// TwinCAT 3 PLC project SPS
// ProgramVersion: 3.1.4024.0
// libraries:
//   Tc2_MC2, * (Beckhoff Automation GmbH)
//   Tc2_Standard, * (Beckhoff Automation GmbH)
//   Tc2_System, * (Beckhoff Automation GmbH)
//   Tc3_IotBase, * (Beckhoff Automation GmbH)
//   Tc3_Module, * (Beckhoff Automation GmbH)
// project tree:
//   DUTs/ eBetriebszustand.TcDUT
//   GVLs/ GVL_PosKinematic.TcGVL, IFC_HW.TcGVL (not stored)
//   / PlcTask.TcTTO
//   POUs/Abfüllmodul/Ampelleuchte/ FB_Ampelstatus.TcPOU (not stored), FB_Blinklicht.TcPOU
//   POUs/Abfüllmodul/ FB_Abfullmodul.TcPOU, FB_Dispenser.TcPOU
//   POUs/Abfüllmodul/Tranport/ FB_Forderband.TcPOU, FB_Transport.TcPOU, FB_TransportA.TcPOU (not stored), FB_TransportE.TcPOU, FB_TransportLogik.TcPOU
//   POUs/Abfüllmodul/Vereinzelung/ FB_EZylinder.TcPOU (not stored), FB_Vereinzelung.TcPOU (not stored)
//   POUs/ FB_Maschinentuer.TcPOU, FB_Testmaschinentuer.TcPOU, MAIN.TcPOU, FUN_linear_Scale.TcPOU
//   POUs/IOT/ FB_MqttClient.TcPOU
//   POUs/Robotermodul/ FB_Roboterablauf.TcPOU, FB_Robotersteuerung.TcPOU, FB_Roboterachsensteuerung.TcPOU
// real-time tasks:
//   TASK PlcTask: cycle T#10ms, priority 20, ADS port 350
// motion (NC):
//   TASK NC-Task 1 SAF: cycle T#2ms, priority 4, ADS port 501
//   TASK NC-Task 1 SVB: cycle T#10ms, priority 8, ADS port 511
//   AXIS Achse_Band (id 1)
//     OtherSettings: AllowMotionCmdToSlave=true
//     encoder EncType=1
//     drive DrvType=5
//       Analog: TorqueSetpointScale=10, ScaleFactorActTorque=0.1
//       TimeComp: TaskDelayCycles=1
//     controller CtrType=1
//       CtrPara: PriorControlFactor=1
//         Observer: BandWidth=20
//   AXIS Achse_Extruder1 (id 2)
//     OtherSettings: AllowMotionCmdToSlave=true
//     encoder EncType=1
//     drive DrvType=5
//       Analog: TorqueSetpointScale=10, ScaleFactorActTorque=0.1
//       TimeComp: TaskDelayCycles=1
//     controller CtrType=1
//       CtrPara: PriorControlFactor=1
//         Observer: BandWidth=20
//   AXIS Achse_Extruder2 (id 3)
//     OtherSettings: AllowMotionCmdToSlave=true
//     encoder EncType=1
//     drive DrvType=5
//       Analog: TorqueSetpointScale=10, ScaleFactorActTorque=0.1
//       TimeComp: TaskDelayCycles=1
//     controller CtrType=1
//       CtrPara: PriorControlFactor=1
//         Observer: BandWidth=20
//   AXIS Achse_Extruder3 (id 4)
//     OtherSettings: AllowMotionCmdToSlave=true
//     encoder EncType=1
//     drive DrvType=5
//       Analog: TorqueSetpointScale=10, ScaleFactorActTorque=0.1
//       TimeComp: TaskDelayCycles=1
//     controller CtrType=1
//       CtrPara: PriorControlFactor=1
//         Observer: BandWidth=20
//   AXIS Roboter_x (id 5)
//     OtherSettings: AllowMotionCmdToSlave=true
//     encoder EncType=1
//       EncPara: ScaleFactorNumerator=1
//         Inc: RefSearchInverse=true, RefSyncInverse=false
//     drive DrvType=5
//       Analog: TorqueSetpointScale=10, ScaleFactorActTorque=0.1
//       TimeComp: TaskDelayCycles=1
//     controller CtrType=1
//       CtrPara: PriorControlFactor=1
//         Observer: BandWidth=20
//   AXIS Roboter_y (id 6)
//     OtherSettings: AllowMotionCmdToSlave=true
//     encoder EncType=1
//       EncPara: ScaleFactorNumerator=1
//         Inc: RefSearchInverse=true, RefSyncInverse=false
//     drive DrvType=5
//       Analog: TorqueSetpointScale=10, ScaleFactorActTorque=0.1
//       TimeComp: TaskDelayCycles=1
//     controller CtrType=1
//       CtrPara: PriorControlFactor=1
//         Observer: BandWidth=20
//   AXIS Roboter_z (id 7)
//     OtherSettings: AllowMotionCmdToSlave=true
//     encoder EncType=1
//       EncPara: ScaleFactorNumerator=1
//         Inc: RefSearchInverse=true, RefSyncInverse=false
//     drive DrvType=5
//       Analog: TorqueSetpointScale=10, ScaleFactorActTorque=0.1
//       TimeComp: TaskDelayCycles=1
//     controller CtrType=1
//       CtrPara: PriorControlFactor=1
//         Observer: BandWidth=20
//   AXIS Roboter_g (id 8)
//     OtherSettings: AllowMotionCmdToSlave=true
//     encoder EncType=1
//       EncPara: ScaleFactorNumerator=1
//     drive DrvType=5
//       Analog: TorqueSetpointScale=10, ScaleFactorActTorque=0.1
//       TimeComp: TaskDelayCycles=1
//     controller CtrType=1
//       CtrPara: PriorControlFactor=1
//         Observer: BandWidth=20
// variable links:
//   SPS/SPS Instance <-> NC-Task 1 SAF/Axes/Achse_Band
//     PlcTask Inputs/IFC_HW.ax_BandMotor.NcToPlc <-> Outputs/ToPlc
//     PlcTask Outputs/IFC_HW.ax_BandMotor.PlcToNc <-> Inputs/FromPlc
//   SPS/SPS Instance <-> NC-Task 1 SAF/Axes/Achse_Extruder1
//     PlcTask Inputs/IFC_HW.ax_Extruder1.NcToPlc <-> Outputs/ToPlc
//     PlcTask Outputs/IFC_HW.ax_Extruder1.PlcToNc <-> Inputs/FromPlc
//   SPS/SPS Instance <-> NC-Task 1 SAF/Axes/Achse_Extruder2
//     PlcTask Inputs/IFC_HW.ax_Extruder2.NcToPlc <-> Outputs/ToPlc
//     PlcTask Outputs/IFC_HW.ax_Extruder2.PlcToNc <-> Inputs/FromPlc
//   SPS/SPS Instance <-> NC-Task 1 SAF/Axes/Achse_Extruder3
//     PlcTask Inputs/IFC_HW.ax_Extruder3.NcToPlc <-> Outputs/ToPlc
//     PlcTask Outputs/IFC_HW.ax_Extruder3.PlcToNc <-> Inputs/FromPlc
//   SPS/SPS Instance <-> NC-Task 1 SAF/Axes/Roboter_g
//     PlcTask Inputs/IFC_HW.ax_ManG.NcToPlc <-> Outputs/ToPlc
//     PlcTask Outputs/IFC_HW.ax_ManG.PlcToNc <-> Inputs/FromPlc
//   SPS/SPS Instance <-> NC-Task 1 SAF/Axes/Roboter_x
//     PlcTask Inputs/IFC_HW.ax_ManX.NcToPlc <-> Outputs/ToPlc
//     PlcTask Outputs/IFC_HW.ax_ManX.PlcToNc <-> Inputs/FromPlc
//   SPS/SPS Instance <-> NC-Task 1 SAF/Axes/Roboter_y
//     PlcTask Inputs/IFC_HW.ax_ManY.NcToPlc <-> Outputs/ToPlc
//     PlcTask Outputs/IFC_HW.ax_ManY.PlcToNc <-> Inputs/FromPlc
//   SPS/SPS Instance <-> NC-Task 1 SAF/Axes/Roboter_z
//     PlcTask Inputs/IFC_HW.ax_ManZ.NcToPlc <-> Outputs/ToPlc
//     PlcTask Outputs/IFC_HW.ax_ManZ.PlcToNc <-> Inputs/FromPlc

CONFIGURATION SPS
    RESOURCE PLC ON TwinCAT3
        TASK PlcTask(INTERVAL := T#10ms, PRIORITY := 20);
        PROGRAM MAIN WITH PlcTask : MAIN;
    END_RESOURCE
END_CONFIGURATION

// ---- DUTs/eBetriebszustand.TcDUT
{attribute 'qualified_only'}
{attribute 'strict'}
TYPE eBetriebszustand :
(
	WARNING,	// Nicht fehlerbehafteter/ungeplanter Stop
	ERROR,		// Fehlerbehafteter Stop
	STOP,		// Geplanter Stop
	OFF,		// Nicht Betriebsbereit
	INIT,		// Herstellung betriebsbereit
	PROD,		// Betrieb
	READY,		// Betriebsbereit
	DONE,		// Betrieb abgeschlosen
	SETUP		// Wartung
);
END_TYPE

// ---- GVLs/GVL_PosKinematic.TcGVL
{attribute 'qualified_only'}
VAR_GLOBAL
	// Home position
	pXhome : REAL := 29;
	pYhome : REAL := 145.5;
	pZhome : REAL := 45;
	
	// Conveyor position
	pXconv : REAL := 29;
	pYconv : REAL := 145.5;
	pZconv : REAL := 130;
	
	// Scale position
	pXscale : REAL := 36;
	pYscale : REAL := 7.5;
	pZscale : REAL := 131.5;
	
	// Heating position
	pXheat : REAL := 218.5;
	pYheat : REAL := 7;
	pZheat : REAL := 159;
	
	// Storage position
	pX1stor : REAL := 107;
	pX2stor : REAL := 158.7;
	pX3stor : REAL := 209.3;
	pX4stor : REAL := 260.3;
	pYstor : REAL := 139;
	pZstor : REAL := 120;
	
	// Z offset height
	pZoff : REAL := 45;
END_VAR

// ---- POUs/MAIN.TcPOU
PROGRAM MAIN
VAR
	fbAbfullmodul : FB_Abfullmodul;
	fbStatusAmpel : FB_Ampelstatus;
	fbRoboter : FB_Roboterablauf;
	fbMqttClient : FB_MqttClient;
END_VAR

fbAbfullmodul(
	bEnable:= IFC_HW.bEnable, 
	bExecute:= IFC_HW.bExecute, 
	eState=> fbStatusAmpel.eState, 
	ax1:= IFC_HW.ax_Extruder1, 
	ax2:= IFC_HW.ax_Extruder2, 
	ax3:= IFC_HW.ax_Extruder3);
	
fbStatusAmpel(
	eState:= , 
	bLightRed=> IFC_HW.bAmpelRot, 
	bLightYellow=> IFC_HW.bAmpelGelb, 
	bLightGreen=> IFC_HW.bAmpelGrun);
	
fbRoboter(bEnable:= IFC_HW.bEnable, bExecute:= IFC_HW.bBandSens4, eState=> );

fbMqttClient();

END_PROGRAM

// ---- POUs/Abfüllmodul/FB_Abfullmodul.TcPOU
FUNCTION_BLOCK FB_Abfullmodul
VAR_INPUT
    bEnable: BOOL;
    bExecute : BOOL;
END_VAR
VAR_OUTPUT
    eState : eBetriebszustand;
END_VAR
VAR
    nState : INT := 0;
    nStation :INT := 0;
    
    fbVereinzelung : FB_Vereinzelung;
    fbTransport : FB_Transport;
    fbDispenser1 : FB_Dispenser;
    fbDispenser2 : FB_Dispenser;
    fbDispenser3 : FB_Dispenser;
	fbEZylinder1: FB_EZylinder;
	fbEZylinder2: FB_EZylinder;
END_VAR
VAR_IN_OUT
    ax1 : AXIS_REF;
	ax2 : AXIS_REF;
	ax3 : AXIS_REF;
END_VAR

fbVereinzelung(
	bEnable:= bEnable, 
	bExecute:= , 
	bSensor1:= IFC_HW.bEinzelSens1, 
	bSensor2:= IFC_HW.bEinzelSens2, 
	bSensor3:= IFC_HW.bEinzelSens3, 
	bSensor4:= IFC_HW.bBandSens1, 
	eState=> , 
	bGate1=> fbEZylinder1.bGate, 
	bGate2=> fbEZylinder2.bGate);
	
fbEZylinder1(bGate:= , bError:= , bR1=> IFC_HW.bR1AKT1, bR2=> IFC_HW.bR2AKT1);
fbEZylinder2(bGate:= , bError:= , bR1=> IFC_HW.bR1AKT2, bR2=> IFC_HW.bR2AKT2);

fbTransport(
	bEnable:= bEnable, 
	bExecute:= , 
	nStation:= nStation, 
	bSens1:= IFC_HW.bBandSens1, 
	bSens2:= IFC_HW.bBandSens2, 
	bSens3:= IFC_HW.bBandSens3, 
	bSens4:= IFC_HW.bBandSens4, 
	eState=> , 
	bStopper1=> IFC_HW.bBandHub1, 
	bStopper2=> IFC_HW.bBandHub2, 
	bStopper3=> IFC_HW.bBandHub3, 
	ax:= IFC_HW.ax_BandMotor);
	
fbDispenser1(
	bEnable:= bEnable, 
	bExecute:= , 
	rDistance:= 100, 
	eState=> , 
	ax:= ax1);

fbDispenser2(
	bEnable:= bEnable, 
	bExecute:= , 
	rDistance:= 100, 
	eState=> , 
	ax:= ax2);

fbDispenser3(
	bEnable:= bEnable, 
	bExecute:= , 
	rDistance:= 100, 
	eState=> , 
	ax:= ax3);

CASE nState OF
	
	0: // OFF
	eState := eBetriebszustand.OFF;
	
	fbVereinzelung.bEnable := FALSE;
	fbTransport.bEnable := FALSE;
	fbDispenser1.bEnable := FALSE;
	fbDispenser2.bEnable := FALSE;
	fbDispenser3.bEnable := FALSE;
	
	fbVereinzelung.bExecute := FALSE;
	fbTransport.bExecute := FALSE;
	fbDispenser1.bExecute := FALSE;
	fbDispenser2.bExecute := FALSE;
	fbDispenser3.bExecute := FALSE;
	
	IF bEnable THEN
		nState:= 10; // INIT
	END_IF
	
	10: // INIT
	eState := eBetriebszustand.INIT;
	
	fbVereinzelung.bEnable := TRUE;
	fbTransport.bEnable := TRUE;
	fbDispenser1.bEnable := TRUE;
	fbDispenser2.bEnable := TRUE;
	fbDispenser3.bEnable := TRUE;
	
	fbVereinzelung.bExecute := FALSE;
	fbTransport.bExecute := FALSE;
	fbDispenser1.bExecute := FALSE;
	fbDispenser2.bExecute := FALSE;
	fbDispenser3.bExecute := FALSE;
	
	IF (fbVereinzelung.eState = eBetriebszustand.READY) AND (fbTransport.eState = eBetriebszustand.READY) AND (fbDispenser1.eState = eBetriebszustand.READY) 
		AND (fbDispenser2.eState = eBetriebszustand.READY) AND (fbDispenser3.eState = eBetriebszustand.READY) THEN
		
		nState := 20; // READY
	END_IF
	
	20: // READY
	eState := eBetriebszustand.READY;
	
	fbVereinzelung.bEnable := TRUE;
	fbTransport.bEnable := TRUE;
	fbDispenser1.bEnable := TRUE;
	fbDispenser2.bEnable := TRUE;
	fbDispenser3.bEnable := TRUE;
	
	IF bExecute THEN
		nState := 30; //Start
	END_IF
	
	30: // PROD - Start
	eState := eBetriebszustand.PROD;
	nStation := 1;
	
	fbVereinzelung.bEnable := TRUE;
	fbTransport.bEnable := TRUE;
	fbDispenser1.bEnable := TRUE;
	fbDispenser2.bEnable := TRUE;
	fbDispenser3.bEnable := TRUE;
	
	fbVereinzelung.bExecute := TRUE;
	fbTransport.bExecute := TRUE;
	fbDispenser1.bExecute := FALSE;
	fbDispenser2.bExecute := FALSE;
	fbDispenser3.bExecute := FALSE;
	
	IF (fbVereinzelung.eState = eBetriebszustand.DONE) AND (fbTransport.eState = eBetriebszustand.DONE)THEN
		nState := 31; // Extruder 1
	END_IF
	
	31: // PROD - Extruder 1
	eState := eBetriebszustand.PROD;
	nStation := 1;

	fbVereinzelung.bExecute := FALSE;
	fbTransport.bExecute := FALSE;
	fbDispenser1.bExecute := TRUE;
	fbDispenser2.bExecute := FALSE;
	fbDispenser3.bExecute := FALSE;
	
	IF fbDispenser1.eState = eBetriebszustand.DONE THEN
		nState := 32; // Bewegung zu Station 2
	END_IF
	
	32: // PROD - Bewegung zu Station 2
	eState := eBetriebszustand.PROD;
	nStation := 2;
	
	fbVereinzelung.bExecute := FALSE;
	fbTransport.bExecute := TRUE;
	fbDispenser1.bExecute := FALSE;
	fbDispenser2.bExecute := FALSE;
	fbDispenser3.bExecute := FALSE;
	
	IF fbTransport.eState = eBetriebszustand.DONE THEN
		nState := 33; //  Extruder 2
	END_IF
	
	33: // PROD - Extruder 2
	eState := eBetriebszustand.PROD;
	nStation := 2;
	
	fbVereinzelung.bExecute := FALSE;
	fbTransport.bExecute := FALSE;
	fbDispenser1.bExecute := FALSE;
	fbDispenser2.bExecute := TRUE;
	fbDispenser3.bExecute := FALSE;
	
	IF fbDispenser2.eState = eBetriebszustand.DONE THEN
		nState := 34; // Bewegung zu Station 3
	END_IF
	
	34: // PROD - Bewegung zu Station 3
	eState := eBetriebszustand.PROD;
	nStation := 3;
	
	fbVereinzelung.bExecute := FALSE;
	fbTransport.bExecute := TRUE;
	fbDispenser1.bExecute := FALSE;
	fbDispenser2.bExecute := FALSE;
	fbDispenser3.bExecute := FALSE;
	
	IF fbTransport.eState = eBetriebszustand.DONE THEN
		nState := 35; // Extruder 3
	END_IF
	
	35: // PROD - Extruder 3
	eState := eBetriebszustand.PROD;
	nStation := 3;
	
	fbVereinzelung.bExecute := FALSE;
	fbTransport.bExecute := FALSE;
	fbDispenser1.bExecute := FALSE;
	fbDispenser2.bExecute := FALSE;
	fbDispenser3.bExecute := TRUE;
	
	IF fbDispenser3.eState = eBetriebszustand.DONE THEN
		nState := 36; // Bewegung zu Abholstation
	END_IF
	
	36: // PROD - Bewegung zu Abholstation
	eState := eBetriebszustand.PROD;
	nStation := 4;
	
	fbVereinzelung.bExecute := FALSE;
	fbTransport.bExecute := TRUE;
	fbDispenser1.bExecute := FALSE;
	fbDispenser2.bExecute := FALSE;
	fbDispenser3.bExecute := FALSE; 
	
	IF fbTransport.eState = eBetriebszustand.DONE THEN
		nState := 40; // DONE
	END_IF
	
	40: // DONE
	eState :=  eBetriebszustand.DONE;
	nStation := 4;
	
	fbTransport.bExecute := False;
	
	IF NOT bExecute THEN
		nState := 20; // READY
	ELSIF nStation = 4 THEN
		nState := 30; // START
	END_IF
	
END_CASE

END_FUNCTION_BLOCK

// ---- POUs/Abfüllmodul/Tranport/FB_Transport.TcPOU
FUNCTION_BLOCK FB_Transport
VAR_INPUT
	bEnable : BOOL;
	bExecute : BOOL;
	nStation : INT;
	
	bSens1 : BOOL;
	bSens2 : BOOL;
	bSens3 : BOOL;
	bSens4 : BOOL;
END_VAR
VAR_OUTPUT
	eState : eBetriebszustand;
	
	bStopper1 : BOOL;
	bStopper2 : BOOL;
	bStopper3 : BOOL;
END_VAR
VAR
	fbTransportE : FB_TransportE;
	fbTransportLogik : FB_TransportLogik;
	fbTransportBand : FB_Forderband;
	fbTransportA : FB_TransportA;
END_VAR
VAR_IN_OUT
    ax : AXIS_REF;
END_VAR

fbTransportE(
	bSens1:= bSens1, 
	bSens2:= bSens2, 
	bSens3:= bSens3, 
	bSens4:= bSens4, 
	bStation1=> , 
	bStation2=> , 
	bStation3=> , 
	bStation4=> );
	
fbTransportLogik(
	eStateE:= fbTransportBand.eState, 
	bEnable:= bEnable, 
	bExecute:= bExecute, 
	nStation:= nStation, 
	bStation1:= fbTransportE.bStation1, 
	bStation2:= fbTransportE.bStation2, 
	bStation3:= fbTransportE.bStation3, 
	bStation4:= fbTransportE.bStation4, 
	eStateA=> eState, 
	bEnableA=> , 
	bExecuteA=> , 
	bHaltA=> , 
	bStop1=> , 
	bStop2=> , 
	bStop3=> );
	
fbTransportBand(
	bEnable:= fbTransportLogik.bEnableA, 
	bExecute:= fbTransportLogik.bExecuteA, 
	bHalt:= fbTransportLogik.bHaltA, 
	eState=> , 
	ax:= ax);
	
fbTransportA(
	bStop1:= fbTransportLogik.bStop1, 
	bStop2:= fbTransportLogik.bStop2, 
	bStop3:= fbTransportLogik.bStop3, 
	bStopper1=> bStopper1, 
	bStopper2=> bStopper2, 
	bStopper3=> bStopper3);

END_FUNCTION_BLOCK

// ---- POUs/Abfüllmodul/Tranport/FB_TransportE.TcPOU
FUNCTION_BLOCK FB_TransportE
VAR_INPUT
	bSens1 : BOOL;
	bSens2 : BOOL;
	bSens3 : BOOL;
	bSens4 : BOOL;
END_VAR
VAR_OUTPUT
	bStation1 : BOOL;
	bStation2 : BOOL;
	bStation3 : BOOL;
	bStation4 : BOOL;
END_VAR
VAR
END_VAR

bStation1 := bSens1;
bStation2 := bSens2;
bStation3 := bSens3;
bStation4 := bSens4;

END_FUNCTION_BLOCK

// ---- POUs/Abfüllmodul/Tranport/FB_TransportLogik.TcPOU
FUNCTION_BLOCK FB_TransportLogik
VAR_INPUT
	eStateE : eBetriebszustand;
	bEnable : BOOL;
	bExecute : BOOL;
	nStation : INT;
	
	bStation1 : BOOL;
	bStation2 : BOOL;
	bStation3 : BOOL;
	bStation4 : BOOL;
END_VAR
VAR_OUTPUT
	eStateA : eBetriebszustand;
	bEnableA : BOOL;
	bExecuteA : BOOL;
	bHaltA : BOOL;
	
	bStop1 : BOOL;
	bStop2 : BOOL;
	bStop3 : BOOL;
END_VAR
VAR
	nState : INT;
END_VAR

CASE nState OF
	0: //OFF
	eStateA := eBetriebszustand.OFF;
	
	bEnableA := FALSE;
	bExecuteA := FALSE;
	bHaltA := FALSE;
	bStop1 := FALSE;
	bStop2 := FALSE;
	bStop3 := FALSE;
	
	IF bEnable THEN
		nState := 1;
	END_IF
	
	1: //INIT
	eStateA := eBetriebszustand.INIT;
	
	bEnableA := TRUE;
	bExecuteA := FALSE;
	bHaltA := FALSE;
	bStop1 := FALSE;
	bStop2 := FALSE;
	bStop3 := FALSE;
	
	IF eStateE = eBetriebszustand.READY THEN
		nState := 2;
	END_IF
	
	2: //READY
	eStateA := eBetriebszustand.READY;
	
	bEnableA := TRUE;
	bExecuteA := FALSE;
	bHaltA := TRUE;
	bStop1 := FALSE;
	bStop2 := FALSE;
	bStop3 := FALSE;
	
	IF bExecute THEN
		nState := 3;
	END_IF
	
	3: //PROD-Förderband start
	eStateA := eBetriebszustand.PROD;
	
	bEnableA := TRUE;
	bExecuteA := TRUE;
	bHaltA := FALSE;
	IF (nStation - 1) = 1 THEN
		bStop1 := TRUE;
		bStop2 := FALSE;
		bStop3 := FALSE;
	ELSIF (nStation - 1) = 2 THEN
		bStop1 := FALSE;
		bStop2 := TRUE;
		bStop3 := FALSE;
	ELSIF (nStation - 1) = 3 THEN
		bStop1 := FALSE;
		bStop2 := FALSE;
		bStop3 := TRUE;
	END_IF
	
	IF bStation1 AND nStation = 1 THEN
		nState := 4;
	ELSIF bStation2 AND nStation = 2 THEN
		nState := 4;
	ELSIF bStation3 AND nStation = 3 THEN
		nState := 4;
	ELSIF bStation4 AND nStation = 4 THEN
		nState := 4;
	END_IF
	
	4: //PROD-Förderband stop
	eStateA := eBetriebszustand.PROD;
	
	bEnableA := TRUE;
	bExecuteA := FALSE;
	bHaltA := TRUE;
	bStop1 := FALSE;
	bStop2 := FALSE;
	bStop3 := FALSE;
	
	IF eStateE = eBetriebszustand.READY THEN
		nState := 5;
	END_IF
	
	5: //DONE
	eStateA := eBetriebszustand.DONE;
	
	IF NOT bExecute THEN
		nState := 2;
	END_IF
END_CASE

END_FUNCTION_BLOCK

// ---- POUs/Abfüllmodul/Tranport/FB_Forderband.TcPOU
FUNCTION_BLOCK FB_Forderband
VAR_INPUT
	// Steuereingang
	bEnable : BOOL;
	bExecute : BOOL;
	bHalt : BOOL;
END_VAR
VAR_OUTPUT
	eState : eBetriebszustand;
END_VAR
VAR
	nState : INT := 0;
	rVelocity : REAL;
	rAccelaration : REAL;
	fbRTrig: R_Trig;
	
	// Motion Blöcke Tc2_Mc2
	mcReset : MC_Reset;
	mcPower : MC_Power;
	mcVelocity : MC_MoveVelocity;
	mcHalt : MC_Halt;
END_VAR
VAR_IN_OUT
	ax : Axis_Ref;
END_VAR

ax.ReadStatus();
mcHalt(
	Axis:= ax, 
	Execute:= , 
	Deceleration:= , 
	Jerk:= , 
	BufferMode:= , 
	Options:= , 
	Done=> , 
	Busy=> , 
	Active=> , 
	CommandAborted=> , 
	Error=> , 
	ErrorID=> );
	
mcReset(
	Axis:= ax, 
	Execute:= , 
	Done=> , 
	Busy=> , 
	Error=> , 
	ErrorID=> );
	
mcPower(
	Axis:= ax, 
	Enable:= , 
	Enable_Positive:= TRUE, 
	Enable_Negative:= , 
	Override:= , 
	BufferMode:= , 
	Options:= , 
	Status=> , 
	Busy=> , 
	Error=> , 
	ErrorID=> );
	
mcVelocity(
	Axis:= ax, 
	Execute:= , 
	Velocity:= 30,
	Acceleration:= 60, 
	Deceleration:= , 
	Jerk:= , 
	Direction:= MC_Positive_Direction, 
	BufferMode:= , 
	Options:= , 
	InVelocity=> , 
	Busy=> , 
	Active=> , 
	CommandAborted=> , 
	Error=> , 
	ErrorID=> );

fbRTrig(CLK:= mcPower.Status, Q=> );
IF fbRTrig.Q THEN
    nState := 0;
END_IF
	
CASE nState OF 
	0: // OFF
	eState := eBetriebszustand.OFF;
	mcPower.Enable := TRUE;
	
	IF mcPower.Status AND bEnable THEN
		nState := 20;
	ELSIF NOT mcPower.Status AND bEnable THEN
		nState := 10;
	END_IF
	
	10: // INIT-Reset
	eState := eBetriebszustand.INIT;
	mcReset.Execute := TRUE;
	mcPower.Enable := FALSE;
	
	IF mcReset.Done THEN
		nState := 11;
		mcReset.Execute := FALSE;
	END_IF
	
	11: // INIT-Power
	eState := eBetriebszustand.INIT;
	mcReset.Execute := FALSE;
	mcPower.Enable := TRUE;
	
	IF mcPower.Status THEN
		nState := 20;
	END_IF
	
	20: // READY
	eState := eBetriebszustand.READY;
	
	IF bExecute THEN
		nState := 30;
	END_IF
	
	30: // PROD-kontinuierliche Bewegung
	eState := eBetriebszustand.PROD;
	mcVelocity.Execute := TRUE;
	mcVelocity.Velocity := 40;
	mcVelocity.Acceleration := 60;
	
	IF bHalt THEN
		nState := 31;
	END_IF
	
	31: // PROD-Halten
	eState := eBetriebszustand.PROD;
	mcVelocity.Execute := FALSE;
	mcHalt.Execute := TRUE;
	mcHalt.Deceleration := 10;
	
	IF mcHalt.Done THEN
		nState := 40;
	END_IF
	
	40: // DONE-Fertig
	eState := eBetriebszustand.DONE;
	mcHalt.Execute := FALSE;
	
	IF NOT bExecute THEN
		nState := 20;
	END_IF
END_CASE

END_FUNCTION_BLOCK

// ---- POUs/Abfüllmodul/FB_Dispenser.TcPOU
FUNCTION_BLOCK FB_Dispenser
VAR_INPUT
    // Steuereingang
    bEnable : BOOL;
    bExecute:BOOL;
    rDistance : REAL;
    
END_VAR
VAR_OUTPUT
    eState : eBetriebszustand;
END_VAR
VAR
    // Motion Blöcke der Tc2_Mc2
    mcPower : MC_Power;
    mcReset : MC_Reset;
    mcRelative : MC_MoveRelative;
	fbRTrig : R_TRIG;
    nState : INT := 0;
END_VAR
VAR_IN_OUT
    ax : AXIS_REF;
END_VAR

ax.ReadStatus();
mcReset(
    Axis:= ax, 
    Execute:= , 
    Done=> , 
    Busy=> , 
    Error=> , 
    ErrorID=> );

mcPower(
    Axis:= ax, 
    Enable:= , 
    Enable_Positive:= TRUE, 
    Enable_Negative:= , 
    Override:= , 
    BufferMode:= , 
    Options:= , 
    Status=> , 
    Busy=> , 
    Error=> , 
    ErrorID=> );

mcRelative(
    Axis:= ax, 
    Execute:= , 
    Distance:= , 
    Velocity:= 30, 
    Acceleration:= 60, 
    Deceleration:= 60, 
    Jerk:= , 
    BufferMode:= , 
    Options:= , 
    Done=> , 
    Busy=> , 
    Active=> , 
    CommandAborted=> , 
    Error=> , 
    ErrorID=> );

fbRTrig(CLK:= mcPower.Status, Q=> );
IF fbRTrig.Q THEN
    nState := 0;
END_IF

CASE nState OF
    0: // OFF
    eState := eBetriebszustand.OFF;

    IF mcPower.Status AND bEnable THEN
        nState := 20; // Ready
    ELSIF NOT mcPower.Status AND bEnable THEN
        nState := 10; // INIT - Reset
    END_IF

    10: // INIT - Reset
     eState := eBetriebszustand.INIT;

     mcReset.Execute := TRUE;
     mcPower.Enable := FALSE;

     IF mcReset.Done THEN
         nState := 11; // INIT - Power
     END_IF

     11: // INIT - Power
     eState := eBetriebszustand.INIT;

     mcPower.Enable := TRUE;
     mcReset.Execute := FALSE;

     IF mcPower.Status THEN
         nState := 20; // Ready
     END_IF

     20: // READY
     eState := eBetriebszustand.READY;

     IF bExecute THEN
         nState := 30; // relative Bewegunng
     END_IF

     30: // PRODE-relative Bewegung
     eState := eBetriebszustand.PROD;

     mcRelative.Execute := TRUE;
     mcRelative.Distance := rDistance;

     IF mcRelative.Done THEN
         nState:= 40; // Done
     END_IF

     40: // DONE
     eState := eBetriebszustand.DONE;
	 mcRelative.Execute := False;

     IF NOT bExecute THEN
         nState := 20; //Ready
     END_IF

END_CASE;

END_FUNCTION_BLOCK

// ---- POUs/Robotermodul/FB_Roboterablauf.TcPOU
FUNCTION_BLOCK FB_Roboterablauf
VAR_INPUT
	bEnable : BOOL;
	bExecute : BOOL;
END_VAR
VAR_OUTPUT
	eState : eBetriebszustand;
END_VAR
VAR
	nState : INT := 0;
	nStation : INT := 1;
	nFlaschenPos : INT := 1;
	fbRobotersteuerung : FB_Robotersteuerung;
	fbTon : TON;
END_VAR

fbRobotersteuerung(
	bEnable:= , 
	bExecute:= , 
	rXpos:= , 
	rYpos:= , 
	rZpos:= , 
	bGclose:= , 
	eState=> );
	
fbTon(IN:= , PT:= T#5S, Q=> , ET=> );
	
CASE nState OF
	0: // OFF
	eState := eBetriebszustand.OFF;
	
	fbRobotersteuerung.bEnable := FALSE;
	
	IF bEnable THEN
		nState := 1;
	END_IF
	
	1: // INIT
	eState := eBetriebszustand.INIT;
	
	fbRobotersteuerung.bEnable := TRUE;
	
	IF fbRobotersteuerung.eState = eBetriebszustand.READY THEN
		nState := 2;
	END_IF
	
	2: // INIT - HomePos
	eState := eBetriebszustand.INIT;
	
	fbRobotersteuerung.rXpos := GVL_PosKinematic.pXhome;
	fbRobotersteuerung.rYpos := GVL_PosKinematic.pYhome;
	fbRobotersteuerung.rZpos := GVL_PosKinematic.pYhome;
	fbRobotersteuerung.bGclose := FALSE;
	fbRobotersteuerung.bExecute := TRUE;
	
	IF fbRobotersteuerung.eState = eBetriebszustand.READY THEN
		fbRobotersteuerung.bExecute := FALSE;
		nState := 3;
	END_IF
	
	3: // READY
	eState := eBetriebszustand.READY;
	
	IF bExecute THEN
		nState := 4;
	END_IF
	
	4: // PROD - PickUp
	eState := eBetriebszustand.PROD;
	
	fbRobotersteuerung.rXpos := GVL_PosKinematic.pXconv;
	fbRobotersteuerung.rYpos := GVL_PosKinematic.pYconv;
	fbRobotersteuerung.rZpos := GVL_PosKinematic.pZconv;
	fbRobotersteuerung.bGclose := TRUE;
	fbRobotersteuerung.bExecute := TRUE;
	fbTon.IN := TRUE;
	IF fbTon.Q THEN nStation := 2; END_IF
	
	IF fbRobotersteuerung.eState = eBetriebszustand.DONE
		AND nStation = 2 THEN
		fbTon.IN := FALSE;
		fbRobotersteuerung.bExecute := FALSE;
		nState := 5;
	END_IF
	
	5: // PROD - Waage
	eState := eBetriebszustand.PROD;
	
	fbRobotersteuerung.rXpos := GVL_PosKinematic.pXscale;
	fbRobotersteuerung.rYpos := GVL_PosKinematic.pYscale;
	fbRobotersteuerung.rZpos := GVL_PosKinematic.pZscale;
	fbRobotersteuerung.bGclose := TRUE;
	fbRobotersteuerung.bExecute := TRUE;
	fbTon.IN := TRUE;
	IF fbTon.Q THEN nStation := 3; END_IF
	
	IF fbRobotersteuerung.eState = eBetriebszustand.DONE 
		AND nStation = 3 THEN
		fbTon.IN := FALSE;
		fbRobotersteuerung.bExecute := FALSE;
		nState := 6;
	END_IF
	
	6: // PROD - Ofen
	eState := eBetriebszustand.PROD;
	
	fbRobotersteuerung.rXpos := GVL_PosKinematic.pXheat;
	fbRobotersteuerung.rYpos := GVL_PosKinematic.pYheat;
	fbRobotersteuerung.rZpos := GVL_PosKinematic.pZheat;
	fbRobotersteuerung.bGclose := TRUE;
	fbRobotersteuerung.bExecute := TRUE;
	fbTon.IN := TRUE;
	IF fbTon.Q THEN nStation := 4; END_IF
	
	IF fbRobotersteuerung.eState = eBetriebszustand.DONE 
		AND nStation = 4 THEN
		fbTon.IN := FALSE;
		fbRobotersteuerung.bExecute := FALSE;
		nState := 7;
	END_IF
	
	7: // PROD - Place
	eState := eBetriebszustand.PROD;
	
	CASE nFlaschenPos OF
	1: fbRobotersteuerung.rXpos := GVL_PosKinematic.pX1stor;
	2: fbRobotersteuerung.rXpos := GVL_PosKinematic.pX2stor;
	3: fbRobotersteuerung.rXpos := GVL_PosKinematic.pX3stor;
	4: fbRobotersteuerung.rXpos := GVL_PosKinematic.pX4stor;
	END_CASE
	fbRobotersteuerung.rYpos := GVL_PosKinematic.pYstor;
	fbRobotersteuerung.rZpos := GVL_PosKinematic.pZstor;
	fbRobotersteuerung.bGclose := FALSE;
	fbRobotersteuerung.bExecute := TRUE;
	fbTon.IN := TRUE;
	IF fbTon.Q THEN nStation := 5; END_IF
	
	IF fbRobotersteuerung.eState = eBetriebszustand.DONE
		AND nStation = 5 THEN
		fbTon.IN := FALSE;
		fbRobotersteuerung.bExecute := FALSE;
		nFlaschenPos := (nFlaschenPos MOD 4) + 1;
		nState := 8;
	END_IF
	
	8: // INIT - HomePos
	eState := eBetriebszustand.INIT;
	
	fbRobotersteuerung.rXpos := GVL_PosKinematic.pXhome;
	fbRobotersteuerung.rYpos := GVL_PosKinematic.pYhome;
	fbRobotersteuerung.rZpos := GVL_PosKinematic.pZhome;
	fbRobotersteuerung.bGclose := FALSE;
	fbRobotersteuerung.bExecute := TRUE;
	fbTon.IN := TRUE;
	IF fbTon.Q THEN nStation := 6; END_IF
	
	IF fbRobotersteuerung.eState = eBetriebszustand.DONE
		AND nStation = 6 THEN
		fbTon.IN := FALSE;
		fbRobotersteuerung.bExecute := FALSE;
		nState := 9;
	END_IF
	
	9: // DONE
	eState := eBetriebszustand.DONE;
	
	IF NOT bExecute	THEN
		fbRobotersteuerung.bExecute := FALSE;
		nState := 3;
	END_IF
	
	
END_CASE

END_FUNCTION_BLOCK

// ---- POUs/Robotermodul/FB_Robotersteuerung.TcPOU
FUNCTION_BLOCK FB_Robotersteuerung
VAR_INPUT
	bEnable : BOOL;
	bExecute : BOOL;
	rXpos : REAL := 29;
	rYpos : REAL := 145.5;
	rZpos : REAL := 45;
	bGclose : BOOL := FALSE;
END_VAR
VAR_OUTPUT
	eState : eBetriebszustand;
END_VAR
VAR
	nState : INT := 0;

	fbRoboterAchseX : FB_Roboterachsensteuerung;
	fbRoboterAchseY : FB_Roboterachsensteuerung;
	fbRoboterAchseZ : FB_Roboterachsensteuerung;
	fbRoboterAchseG : FB_Roboterachsensteuerung;
END_VAR

fbRoboterAchseX(
	bEnable:= bEnable, 
	bExecute:= , 
	rPosition:= , 
	rVelocity:= 1000, 
	rAccelaration:= , 
	bRefSens:= IFC_HW.bManEndXmin, 
	eState=> , 
	ax:= IFC_HW.ax_ManX);
	
fbRoboterAchseY(
	bEnable:= bEnable, 
	bExecute:= , 
	rPosition:= , 
	rVelocity:= 1000, 
	rAccelaration:= , 
	bRefSens:= IFC_HW.bManEndYmin, 
	eState=> , 
	ax:= IFC_HW.ax_ManY);
	
fbRoboterAchseZ(
	bEnable:= bEnable, 
	bExecute:= , 
	rPosition:= , 
	rVelocity:= 1000, 
	rAccelaration:= , 
	bRefSens:= IFC_HW.bManEndZmin, 
	eState=> , 
	ax:= IFC_HW.ax_ManZ);

fbRoboterAchseG(
	bEnable:= bEnable, 
	bExecute:= , 
	rPosition:= , 
	rVelocity:= 1000, 
	rAccelaration:= , 
	bRefSens:= IFC_HW.bManEndGmin, 
	eState=> , 
	ax:= IFC_HW.ax_ManG);
		
CASE nState OF
	0: // OFF
	eState := eBetriebszustand.OFF;
	
	fbRoboterAchseX.bEnable := FALSE;
	fbRoboterAchseY.bEnable := FALSE;
	fbRoboterAchseZ.bEnable := FALSE;
	fbRoboterAchseG.bEnable := FALSE;
	
	IF bEnable THEN
		nState := 10;
	END_IF
	
	10: // INIT
	eState := eBetriebszustand.INIT;
	
	fbRoboterAchseX.bEnable := TRUE;
	fbRoboterAchseY.bEnable := TRUE;
	fbRoboterAchseZ.bEnable := TRUE;
	fbRoboterAchseG.bEnable := TRUE;
	
	IF (fbRoboterAchseX.eState = eBetriebszustand.READY) AND (fbRoboterAchseY.eState = eBetriebszustand.READY) AND 
	   (fbRoboterAchseZ.eState = eBetriebszustand.READY) AND (fbRoboterAchseG.eState = eBetriebszustand.READY) THEN   
	   nState := 20;
	END_IF
	
	20: // READY
	eState := eBetriebszustand.READY;
	
	IF bExecute THEN
		nState := 30;
	END_IF
	
	30: // PROD-ZAchse hoch
	eState := eBetriebszustand.PROD;
	IFC_HW.bManBrakeZ := TRUE;
	fbRoboterAchseZ.rPosition := GVL_PosKinematic.pZoff;
	fbRoboterAchseZ.bExecute := TRUE;
	
	IF fbRoboterAchseZ.eState = eBetriebszustand.DONE THEN
		IFC_HW.bManBrakeZ := FALSE;
		fbRoboterAchseZ.bExecute := FALSE;
		nstate := 31;
	END_IF
	
	31: // PROD-XYAchse bewegen
	eState := eBetriebszustand.PROD;
	fbRoboterAchseX.rPosition := rXpos;
	fbRoboterAchseX.bExecute := TRUE;
	fbRoboterAchseY.rPosition := rYpos;
	fbRoboterAchseY.bExecute := TRUE;

	
	IF (fbRoboterAchseX.eState = eBetriebszustand.DONE) AND (fbRoboterAchseY.eState = eBetriebszustand.DONE) THEN
		fbRoboterAchseX.bExecute := FALSE;
		fbRoboterAchseY.bExecute := FALSE;
		nstate := 32;
	END_IF
	
	32: // PROD-ZAchse bewegen
	eState := eBetriebszustand.PROD;
	IFC_HW.bManBrakeZ := TRUE;
	fbRoboterAchseZ.rPosition := rZpos;
	fbRoboterAchseZ.bExecute := TRUE;
	
	IF fbRoboterAchseZ.eState = eBetriebszustand.DONE THEN
		IFC_HW.bManBrakeZ := FALSE;
		fbRoboterAchseZ.bExecute := FALSE;
		nstate := 33;
	END_IF
	
	33: // PROD-GAchse bewegen
	eState := eBetriebszustand.PROD;
	IF bGclose THEN
		fbRoboterAchseG.rPosition := 8.8;
		fbRoboterAchseG.bExecute := TRUE;
		IFC_HW.bGripperClosed := TRUE;
	ELSE
		fbRoboterAchseG.rPosition := 7;
		fbRoboterAchseG.bExecute := TRUE;
		IFC_HW.bGripperClosed := FALSE;
	END_IF
		
	IF fbRoboterAchseG.eState = eBetriebszustand.DONE THEN
		fbRoboterAchseG.bExecute := FALSE;
		nstate := 40;
	END_IF
	
	40: // DONE
	eState := eBetriebszustand.DONE;
	
	IF NOT bExecute THEN
		nState := 20; // READY
	END_IF
END_CASE

END_FUNCTION_BLOCK

// ---- POUs/Robotermodul/FB_Roboterachsensteuerung.TcPOU
FUNCTION_BLOCK FB_Roboterachsensteuerung
VAR_INPUT
	// Steuereingang
	bEnable : BOOL;
	bExecute : BOOL;
	rPosition : REAL;
	rVelocity : REAL := 30;
	rAccelaration : REAL := 60;
	bRefSens: BOOL;
END_VAR
VAR_OUTPUT
	eState : eBetriebszustand;
END_VAR
VAR
	nState : INT := 0;
	
	// Motion Blöcke Tc2_Mc2
	mcReset : MC_Reset;
	mcPower : MC_Power;
	mcHome : MC_Home;
	mcAbsolute : MC_MoveAbsolute;
	
	fbRTrig: R_TRIG;
	
END_VAR
VAR_IN_OUT
	ax : AXIS_REF;
END_VAR

ax.ReadStatus();
	
mcReset(
	Axis:= ax, 
	Execute:= , 
	Done=> , 
	Busy=> , 
	Error=> , 
	ErrorID=> );
	
mcPower(
	Axis:= ax, 
	Enable:= bEnable, 
	Enable_Positive:= TRUE, 
	Enable_Negative:= TRUE, 
	Override:= , 
	BufferMode:= , 
	Options:= , 
	Status=> , 
	Busy=> , 
	Error=> , 
	ErrorID=> );

mcHome(
	Axis:= ax, 
	Execute:= , 
	Position:= , 
	HomingMode:= , 
	BufferMode:= , 
	Options:= , 
	bCalibrationCam:= NOT bRefSens, 
	Done=> , 
	Busy=> , 
	Active=> , 
	CommandAborted=> , 
	Error=> , 
	ErrorID=> );
	
mcAbsolute(
	Axis:= ax, 
	Execute:=, 
	Position:= rPosition, 
	Velocity:= rVelocity, 
	Acceleration:= rAccelaration, 
	Deceleration:= rAccelaration, 
	Jerk:= , 
	BufferMode:= , 
	Options:= , 
	Done=> , 
	Busy=> , 
	Active=> , 
	CommandAborted=> , 
	Error=> , 
	ErrorID=> );

CASE nState OF
	0: // OFF
	eState := eBetriebszustand.OFF;
	
	mcPower.Enable := TRUE;
	mcReset.Execute := FALSE;
	
	IF bEnable THEN
		nState := 10; // INIT-Reset
	END_IF
	
	10: // INIT-Reset
	eState := eBetriebszustand.INIT;
		
	mcPower.Enable := FALSE;
	mcReset.Execute := TRUE;
	
	IF mcReset.Done THEN
		nState := 11; // INIT-Power
	END_IF
	
	11: // INIT-Power
	eState := eBetriebszustand.INIT;
		
	mcPower.Enable := TRUE;
	mcReset.Execute := FALSE;
	
	IF mcPower.Status AND NOT ax.Status.Homed THEN
		nState := 12; // INIT-Home
	ELSIF mcPower.Status AND ax.Status.Homed THEN
		nState := 20; // READY
	END_IF
	
	12: // INIT-Home
	eState := eBetriebszustand.INIT;
	
	mcHome.Execute := TRUE;
	
	IF mcHome.Done THEN
		mcHome.Execute := FALSE;
		nState := 20; // READY
	END_IF
	
	20: // READY
	eState := eBetriebszustand.READY;
	
	IF bExecute THEN
		nState := 30; // PROD-Bewegen
	END_IF
	
	30: // PROD-Bewegen
	eState := eBetriebszustand.PROD;
	
	mcAbsolute.Position := rPosition;
	mcAbsolute.Execute := TRUE;
	
	IF mcAbsolute.Done THEN
		mcAbsolute.Execute := False;
		nState := 40; // DONE
	END_IF
	
	40: // DONE
	eState := eBetriebszustand.DONE;
	
	IF NOT bExecute THEN
		nState := 20; // READY
	END_IF
	
END_CASE

END_FUNCTION_BLOCK

// ---- POUs/IOT/FB_MqttClient.TcPOU
FUNCTION_BLOCK FB_MqttClient
VAR_INPUT
END_VAR
VAR_OUTPUT
END_VAR
VAR
    fbMqttClient : FB_IotMqttClient;
    sTopicToPublish: STRING(255) := 'Temperature'; 	// MQTT topic for temperature
    sMessageToPublish: STRING(255); 				// Message buffer
    tmrSendMessageInterval: TON := (PT := T#1S); 	// Interval timer for publishing
    ai_RoomTemperature: INT := 1; 					// Room temperature from thermocouple
	is_init : BOOL := FALSE;
END_VAR

fbMqttClient.sClientId:= 'Publishing PLC';
fbMqttClient.sHostName:= '158.180.44.197';
fbMqttClient.nHostPort:= 1883;
fbMqttClient.sTopicPrefix:= 'aut/apt-get rekt/'; 
fbMqttClient.sUserName:= 'bobm';
fbMqttClient.sUserPassword:= 'letmein';

fbMqttClient.Execute(bConnect := TRUE);

//METH_Publish('$$groupname', 'apt-get rekt');
//METH_Publish('names', 'Erdogan - Holzmann - Jolfai');
//METH_Publish('bEnable', bool_to_string(IFC_HW.bEnable));
METH_Publish('bEnable/$$unit', 'BOOL');

METHOD METH_Publish : BOOL
VAR_INPUT
	sTopicToPublish : STRING;
	sMessageToPublish : STRING;
END_VAR
IF fbMqttClient.bConnected THEN
    tmrSendMessageInterval(IN := TRUE);
    IF tmrSendMessageInterval.Q THEN
        tmrSendMessageInterval(IN := FALSE);
        //sMessageToPublish := REAL_TO_STRING(ai_RoomTemperature / 10.0);

        fbMqttClient.Publish(
            sTopic := sTopicToPublish,
            pPayload := ADR(sMessageToPublish),
            nPayloadSize := LEN(sMessageToPublish) + 1,
            eQoS := TcIotMqttQos.AtMostOnceDelivery,
            bRetain := TRUE,
            bQueue := TRUE
        );
    END_IF
END_IF
END_METHOD

END_FUNCTION_BLOCK

// ---- POUs/Abfüllmodul/Ampelleuchte/FB_Blinklicht.TcPOU
FUNCTION_BLOCK FB_Blinklicht
VAR_INPUT
	bEinAus		: BOOL;
	tPeriode	: TIME := T#1S;
END_VAR
VAR_OUTPUT
	bBlink		: BOOL;
END_VAR
VAR
	fbTon		: TON;
END_VAR

fbTon(IN:=bEinAus AND NOT fbTon.Q , PT:=tPeriode , Q=> , ET=> );

IF fbTON.ET <= fbTON.PT/2 THEN
	bBlink := FALSE;
ELSE
	bBlink := TRUE;
END_IF

IF NOT bEinAus THEN
	bBlink := FALSE;
END_IF

END_FUNCTION_BLOCK

// ---- POUs/FB_Maschinentuer.TcPOU
FUNCTION_BLOCK FB_Maschinentuer
VAR_INPUT
	// Sensoreingang
	bDoorO	: BOOL;
	bDoorC	: BOOL;
	// Steuereingang
	bEnable	: BOOL;
	bOpen 	: BOOL;
	bClose 	: BOOL;
END_VAR
VAR_OUTPUT
	// Aktor Ausgang
	bVentil	: BOOL;
	// Zustände
	bError	: BOOL;
END_VAR
VAR
	nState : INT;
END_VAR

CASE nState OF
	0: // Tür geschlossen
	// Ausgänge setzen
	bVentil := TRUE;
	
	// Übergangsbedingung
	IF NOT bDoorC AND bEnable THEN
		nState := 3; // Tür schließen
	ELSIF bOpen THEN
		nState := 1; // Tür öffnen
	END_IF
	
	1: // Tür öffen
	// Ausgänge setzen
	bVentil := FALSE;
	
	// Übergangsbedingung
	IF NOT bDoorO THEN
		nState := nState + 1; // Tür geöffnet
	END_IF
	
	2: // Tür offen
	// Ausgänge setzen
	bVentil := FALSE;
	
	// Übergangsbedingung
	IF bClose AND bEnable THEN
		nState := nState + 1; // Tür schließen
	END_IF
	
	3: // Tür schließen
	// Ausgänge setzen
	bVentil := TRUE;
	
	// Übergangsbedingung
	IF NOT bDoorC THEN
		nState := 0; // Tür geöffnet
	END_IF
END_CASE

END_FUNCTION_BLOCK

// ---- POUs/FB_Testmaschinentuer.TcPOU
FUNCTION_BLOCK FB_Testmaschinentuer
VAR_INPUT
	bVentil	: BOOL;
END_VAR
VAR_OUTPUT
	bDoorC	: BOOL;
	bDoorO	: BOOL;
END_VAR
VAR
	fbTon_O	: TON;
	fbTon_C	: TON;
	tDuration : TIME := T#5S;
END_VAR

fbTon_C(IN:= bVentil, PT:= tDuration, Q=> , ET=> );
fbTon_O(IN:= NOT bVentil, PT:= tDuration, Q=> , ET=> );

IF bVentil THEN
	bDoorO := FALSE;
	
	IF fbTon_C.Q THEN
		bDoorC := TRUE;
	END_IF
ELSIF NOT bVentil THEN
	bDoorC := FALSE;

	IF fbTon_O.Q THEN
		bDoorO := TRUE;
	END_IF
END_IF

END_FUNCTION_BLOCK

// ---- POUs/FUN_linear_Scale.TcPOU
FUNCTION FUN_linear_Scale : REAL
VAR_INPUT
	ix : REAL;
	ixmax : REAL;
	ixmin : REAL;
	rymax : REAL;
	rymin : REAL;
END_VAR
VAR
	rk : REAL := 0;
	rd : REAL := 0;
END_VAR

rk := (rymax - rymin) / (ixmax - ixmin);
rd := rymin - rk + rd;

FUN_linear_Scale := rk * ix + rd;

IF FUN_linear_Scale > rymax THEN
	FUN_linear_Scale := rymax;
ELSIF FUN_linear_Scale < rymin THEN
	FUN_linear_Scale := rymin;
END_IF

END_FUNCTION
